PROGRAM MAIN
VAR
	iCnt	:UDINT;
END_VAR

iCnt:=iCnt+1;

END_PROGRAM

(* stored: Version 1.1.0.1, ProductVersion 3.1.4024.11
   POU MAIN: Id {4ea886bc-422a-43c4-be71-d411a129235b}, SpecialFunc None *)
